TYPE ST_ErrorEvents :
	STRUCT
		(* Errors *)
		PressureDiffEvaporatorTooHigh		: ST_Event := (eventType := E_EventType.PressureDiffEvaporatorTooHigh, isSelfHealing:=FALSE, severity:= E_Severity.Error, message := 'Druckdifferenz am Verdampfer zu hoch. Einfriergefahr');  
		EvaporatingTemperatureTooLow		: ST_Event := (eventType := E_EventType.EvaporatingTemperatureTooLow, isSelfHealing:=TRUE, severity:= E_Severity.Error, message := 'Autrittstemperatur zu niedrig');  
		EvaporatingFlowRateTooLow			: ST_Event := (eventType := E_EventType.EvaporatingFlowRateTooLow, isSelfHealing:=TRUE, severity:= E_Severity.Error, message := 'Durchflussmenge zu niedrig');  
		LowPressureRefrigerationThermostat	: ST_Event := (eventType := E_EventType.LowPressureRefrigerationThermostat, isSelfHealing:=FALSE, severity:= E_Severity.Error, message := 'Thermostat: Niederdruck zu niedrig');  
		HighPressureRefrigerationThermostat	: ST_Event := (eventType := E_EventType.HighPressureRefrigerationThermostat, isSelfHealing:=FALSE, severity:= E_Severity.Error, message := 'Thermostat: Hochdruck zu hoch');  
		MotorProtectionTriggered			: ST_Event := (eventType := E_EventType.MotorProtectionTriggered, isSelfHealing:=FALSE, severity:= E_Severity.Error, message := 'Motorschutzschalter hat ausgelöst');  
		ExpansionValveTriggered				: ST_Event := (eventType := E_EventType.ExpansionValveTriggered, isSelfHealing:=FALSE, severity:= E_Severity.Error, message := 'Expansionsventil ausgelöst');
		IntermediateCircuitFlowRateTooLow	: ST_Event := (eventType := E_EventType.IntermediateCircuitFlowRateTooLow, isSelfHealing:=TRUE, severity:= E_Severity.Error, message := 'Sole Durchflussmenge im Zwischenkreis zu niedrig');
		LowPressureRefrigerationCalc		: ST_Event := (eventType := E_EventType.LowPressureRefrigerationCalc, isSelfHealing:=FALSE, severity:= E_Severity.Error, message := 'Sensor: Niederdruck zu niedrig');  
		TemperatureSourceWaterOutMinTooLow	: ST_Event := (eventType := E_EventType.TemperatureSourceWaterOutMinTooLow, isSelfHealing:=TRUE, severity:= E_Severity.Error, message := 'Quellwasser-Autrittstemperatur zu niedrig. Einfriergefahr');  
	END_STRUCT
END_TYPE

(* stored: Version 1.1.0.1
   DUT ST_ErrorEvents: Id {7cb6974c-5521-4862-b356-e11d5f4dfdd9} *)
